FUNCTION_BLOCK CoE_property_udint EXTENDS CoE_property
VAR_INPUT
END_VAR
VAR_OUTPUT
END_VAR
VAR
	_value : UDINT;
END_VAR

SUPER^();

PROPERTY dataTypeSize : UINT
GET
dataTypeSize := SIZEOF(_value);
END_GET
END_PROPERTY

METHOD get_value : BOOL
VAR_OUTPUT
	value : UDINT ;
	errId : UDINT;
END_VAR
IF init_done THEN
	value := _value;
	get_value := TRUE;
ELSE
	errId := 2;
	get_value := FALSE;
END_IF
END_METHOD

METHOD handle_read_callback : BOOL
VAR_INPUT
	pt_buffer : POINTER TO CoE_buffer_type_cast_union;
	errId : UDINT;
END_VAR

_value := pt_buffer^.value_udint;
_init_done:=TRUE;
_read_errId:=errId;
END_METHOD

METHOD set_value : BOOL
VAR_INPUT
	value : UDINT ;
END_VAR
_valueToWrite.value_udint := value;
IF THIS^._I_CoE_communication_handler <> 0 THEN 
	THIS^._I_CoE_communication_handler.add_write_request(THIS^);
ELSE
	errId:=1;
END_IF
END_METHOD

END_FUNCTION_BLOCK

(* stored: Version 1.1.0.1, ProductVersion 3.1.4024.6
   POU CoE_property_udint: Id {28879696-492e-0c7b-17c6-1cd73028e6f2}, SpecialFunc None
   Property dataTypeSize: Id {0370a145-50d5-0ca1-14e3-05c8cf986572}
   Get Get: Id {ef38bd02-4041-093a-36fe-4d03fbeff813}
   Method get_value: Id {9d25b38a-87d5-0d3c-09fd-a0e8f1b5312d}
   Method handle_read_callback: Id {727d44a0-4f30-087c-091b-6bb6f8be6e33}
   Method set_value: Id {71480052-6765-0c3a-2bdb-c0fb9e05f7e1} *)
